# EPICS substitutions: ioc/SRS300App/Db/devSRS_PS325_neg.substitutions
##########################################################################
# Copyright (c) 2012 Lawrence Berkeley National Laboratory, Accelerator
# Technology Group, Engineering Division
# This code is distributed subject to a Software License Agreement found
# in file LICENSE that is included with this distribution.
##########################################################################

#
# SRS PS325 with polarity switch in - position
#
file devSRS_PS3xx.template
{
  { VMIN="-2500", VMAX="0", IMIN="-10.5e-3", IMAX="0" }
}
